// Mitsubishi GX Works2 project: Prototype   PLC: FX3U/FX3UC

PROGRAM MAIN
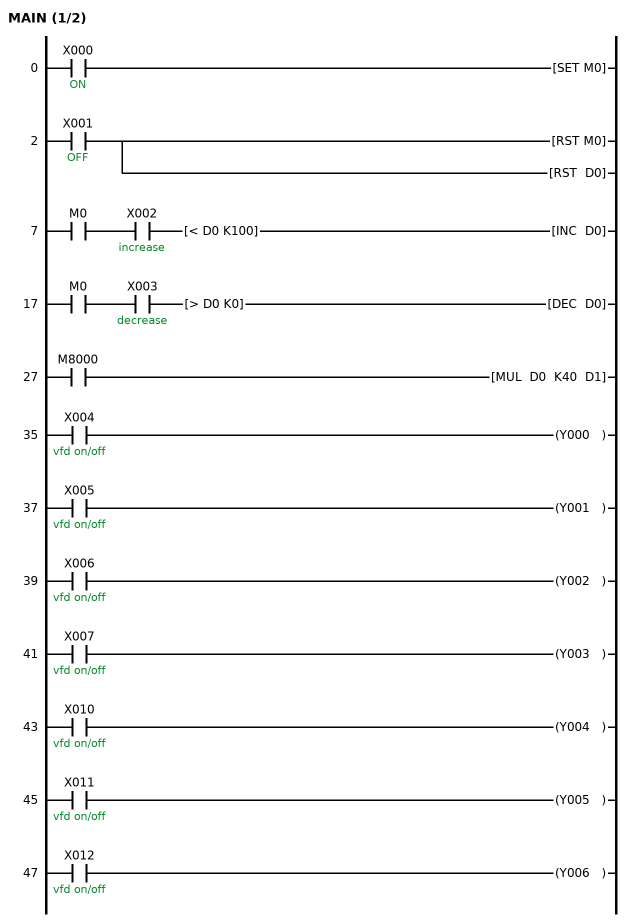
0     LD      X000  ; ON
      SET     M0
2     LD      X001  ; OFF
      RST     M0
      RST     D0
7     LD      M0
      AND     X002  ; increase
      AND<    D0 K100
      INC     D0
17    LD      M0
      AND     X003  ; decrease
      AND>    D0 K0
      DEC     D0
27    LD      M8000
      MUL     D0 K40 D1
35    LD      X004  ; vfd on/off
      OUT     Y000
37    LD      X005  ; vfd on/off
      OUT     Y001
39    LD      X006  ; vfd on/off
      OUT     Y002
41    LD      X007  ; vfd on/off
      OUT     Y003
43    LD      X010  ; vfd on/off
      OUT     Y004
45    LD      X011  ; vfd on/off
      OUT     Y005
47    LD      X012  ; vfd on/off
      OUT     Y006
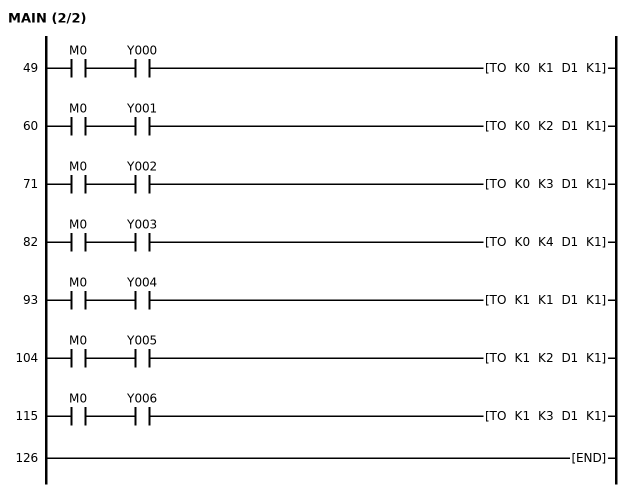
49    LD      M0
      AND     Y000
      TO      K0 K1 D1 K1
60    LD      M0
      AND     Y001
      TO      K0 K2 D1 K1
71    LD      M0
      AND     Y002
      TO      K0 K3 D1 K1
82    LD      M0
      AND     Y003
      TO      K0 K4 D1 K1
93    LD      M0
      AND     Y004
      TO      K1 K1 D1 K1
104   LD      M0
      AND     Y005
      TO      K1 K2 D1 K1
115   LD      M0
      AND     Y006
      TO      K1 K3 D1 K1
126   END
END_PROGRAM
